(* Schneider Machine Expert - Basic project Tank_Level_RTD_1m_TM221CE40T, file version 3.0.0.0 *)
(* ProjectInformations: Name=New project *)

HARDWARE
  Cpu 0: TM221CE40T
  ModuleExtensionObject 0: TM3TI4/G
  EthernetConfiguration: NetworkName=M221, IpAllocationMode=FixedAddress, IpAddress=0.0.0.0, SubnetMask=0.0.0.0
  SerialLineConfiguration: Baud=Baud19200, Parity=ParityEven, DataBits=DataBits8, StopBits=StopBits1, PhysicalMedium=PhysicalMediumRs485, TransmissionMode=TransmissionModeModbusRtu, SlaveId=1, Addressing=SlaveAddressing
  MastTask: UsePeriodScanMode=false, PeriodScan=100
  FastTask: Period=255
  CpuBehavior: StartingMode=StartAsPreviousState, AutoSaveRamOnEeprom=true, WatchdogPeriod=250

SYMBOLS  (address, symbol, comment, settings)
  %M0       SYSTEM_READY
  %M1       TANK_FULL
  %M2       TANK_EMPTY
  %M3       FILLING_MODE
  %M4       DRAINING_MODE
  %M5       INLET_VLV_ALARM
  %M6       OUTLET_VLV_ALARM
  %M10      ANY_ALARM
  %S0       SB_COLDSTART  "Indicates or executes a cold start (data initialized to default values)"
  %S1       SB_WARMSTART  "Indicates there was a warm start with data backup"
  %MF102    HMI_TANK_LITERS  "HMI Tag: Tank volume in liters (0.0-1000.0) - scaled from %MW100"
  %MF103    HMI_TEMPERATURE  "HMI Tag: Temperature in degrees C - scaled from %MW101"
  %MF104    HMI_LEVEL_PERCENT  "HMI Tag: Level percentage (0.0-100.0) - calculated from %MF102"
  %TM1        [Preset=10, Base=OneSecond]
  %TM2        [Preset=5, Base=OneSecond]
  %TM3        [Preset=5, Base=OneSecond]
  %I0.0     EMERGENCY_PB
  %IW0.0      [Type=Type_0_10V, Scope=Scope_Normal, Minimum=0, Maximum=1000]
  %IW1.0    RTD_TEMP  [Type=Type_PT100, Scope=Scope_Standard, Minimum=-200, Maximum=850]

POU Tank Level Control
  (* SectionNumber=0 *)

// Rung 0: Reset_HMI
// Reset HMI floats on cold/warm start to prevent stale data display
  LD %S0                  (* SB_COLDSTART - Cold start *)
  OR %S1                  (* SB_WARMSTART - Warm start *)
  [ %MF102 := 0.0 ]       (* HMI_TANK_LITERS - Reset HMI Tank Liters *)
  [ %MF103 := 0.0 ]       (* HMI_TEMPERATURE - Reset HMI Temperature *)
  [ %MF104 := 0.0 ]       (* HMI_LEVEL_PERCENT - Reset HMI Level Percent *)
  // as ST:
  //   IF SB_COLDSTART OR SB_WARMSTART THEN HMI_TANK_LITERS := 0.0; END_IF;
  //   IF SB_COLDSTART OR SB_WARMSTART THEN HMI_TEMPERATURE := 0.0; END_IF;
  //   IF SB_COLDSTART OR SB_WARMSTART THEN HMI_LEVEL_PERCENT := 0.0; END_IF;
  (* the ladder stored for this rung does not match its IL; not drawn *)

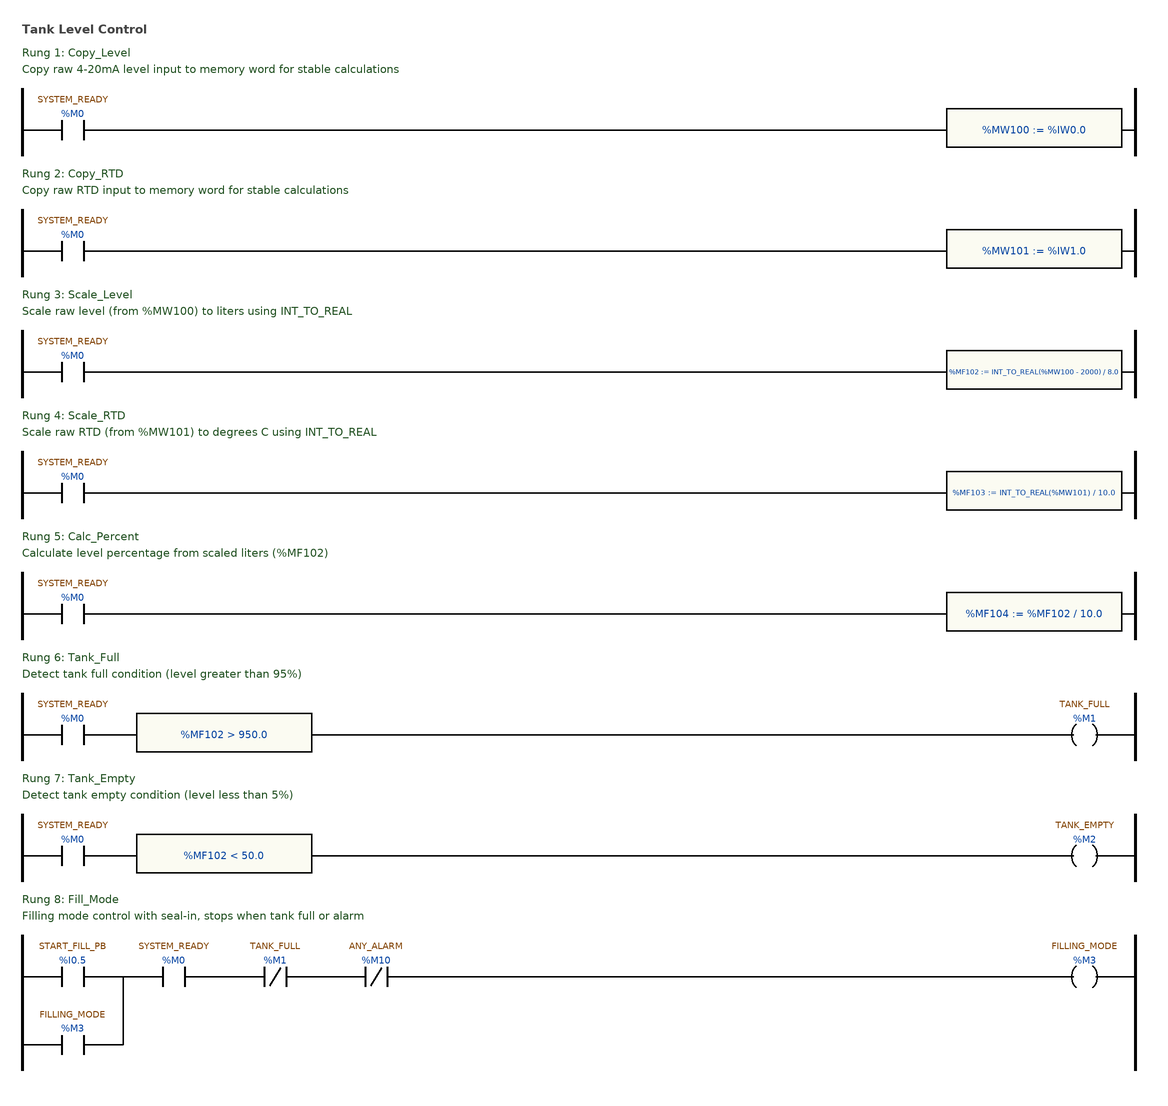

// Rung 1: Copy_Level
// Copy raw 4-20mA level input to memory word for stable calculations
  LD %M0                  (* SYSTEM_READY - System Ready *)
  [ %MW100 := %IW0.0 ]    (* Copy raw level to memory word *)
  // %M0: System Ready
  // as ST:
  //   IF SYSTEM_READY THEN %MW100 := %IW0.0; END_IF;

// Rung 2: Copy_RTD
// Copy raw RTD input to memory word for stable calculations
  LD %M0                  (* SYSTEM_READY - System Ready *)
  [ %MW101 := %IW1.0 ]    (* RTD_TEMP - Copy raw RTD to memory word *)
  // %M0: System Ready
  // as ST:
  //   IF SYSTEM_READY THEN %MW101 := RTD_TEMP; END_IF;

// Rung 3: Scale_Level
// Scale raw level (from %MW100) to liters using INT_TO_REAL
  LD %M0                  (* SYSTEM_READY - System Ready *)
  [ %MF102 := INT_TO_REAL(%MW100 - 2000) / 8.0 ](* HMI_TANK_LITERS - Scale 4-20mA to 0-1000.0 liters *)
  // %M0: System Ready
  // as ST:
  //   IF SYSTEM_READY THEN HMI_TANK_LITERS := INT_TO_REAL(%MW100 - 2000) / 8.0; END_IF;

// Rung 4: Scale_RTD
// Scale raw RTD (from %MW101) to degrees C using INT_TO_REAL
  LD %M0                  (* SYSTEM_READY - System Ready *)
  [ %MF103 := INT_TO_REAL(%MW101) / 10.0 ](* HMI_TEMPERATURE - Scale raw RTD to degrees C *)
  // %M0: System Ready
  // as ST:
  //   IF SYSTEM_READY THEN HMI_TEMPERATURE := INT_TO_REAL(%MW101) / 10.0; END_IF;

// Rung 5: Calc_Percent
// Calculate level percentage from scaled liters (%MF102)
  LD %M0                  (* SYSTEM_READY - System Ready *)
  [ %MF104 := %MF102 / 10.0 ](* HMI_LEVEL_PERCENT, HMI_TANK_LITERS - 0-1000 liters to 0-100.0 percent *)
  // %M0: System Ready
  // as ST:
  //   IF SYSTEM_READY THEN HMI_LEVEL_PERCENT := HMI_TANK_LITERS / 10.0; END_IF;

// Rung 6: Tank_Full
// Detect tank full condition (level greater than 95%)
  LD %M0                  (* SYSTEM_READY - System Ready *)
  AND [ %MF102 > 950.0 ]  (* HMI_TANK_LITERS - Level > 95% *)
  ST %M1                  (* TANK_FULL - Tank Full *)
  // %M0: System Ready
  // %M1: Tank Full Flag
  // as ST:
  //   TANK_FULL := SYSTEM_READY AND HMI_TANK_LITERS > 950.0;

// Rung 7: Tank_Empty
// Detect tank empty condition (level less than 5%)
  LD %M0                  (* SYSTEM_READY - System Ready *)
  AND [ %MF102 < 50.0 ]   (* HMI_TANK_LITERS - Level less than 5% *)
  ST %M2                  (* TANK_EMPTY - Tank Empty *)
  // %M0: System Ready
  // %M2: Tank Empty Flag
  // as ST:
  //   TANK_EMPTY := SYSTEM_READY AND HMI_TANK_LITERS < 50.0;

// Rung 8: Fill_Mode
// Filling mode control with seal-in, stops when tank full or alarm
  LD %I0.5                (* Start Fill Button *)
  OR %M3                  (* FILLING_MODE - Seal-in *)
  AND %M0                 (* SYSTEM_READY - System Ready *)
  ANDN %M1                (* TANK_FULL - Not Tank Full *)
  ANDN %M10               (* ANY_ALARM - No Alarm *)
  ST %M3                  (* FILLING_MODE - Filling Mode *)
  // %I0.5: Start Fill Button
  // %M0: System Ready
  // %M1: Not Tank Full
  // %M10: No Alarm
  // %M3: Filling Mode
  // %M3: Seal-in
  // as ST:
  //   FILLING_MODE := (%I0.5 OR FILLING_MODE) AND SYSTEM_READY AND NOT TANK_FULL AND NOT ANY_ALARM;

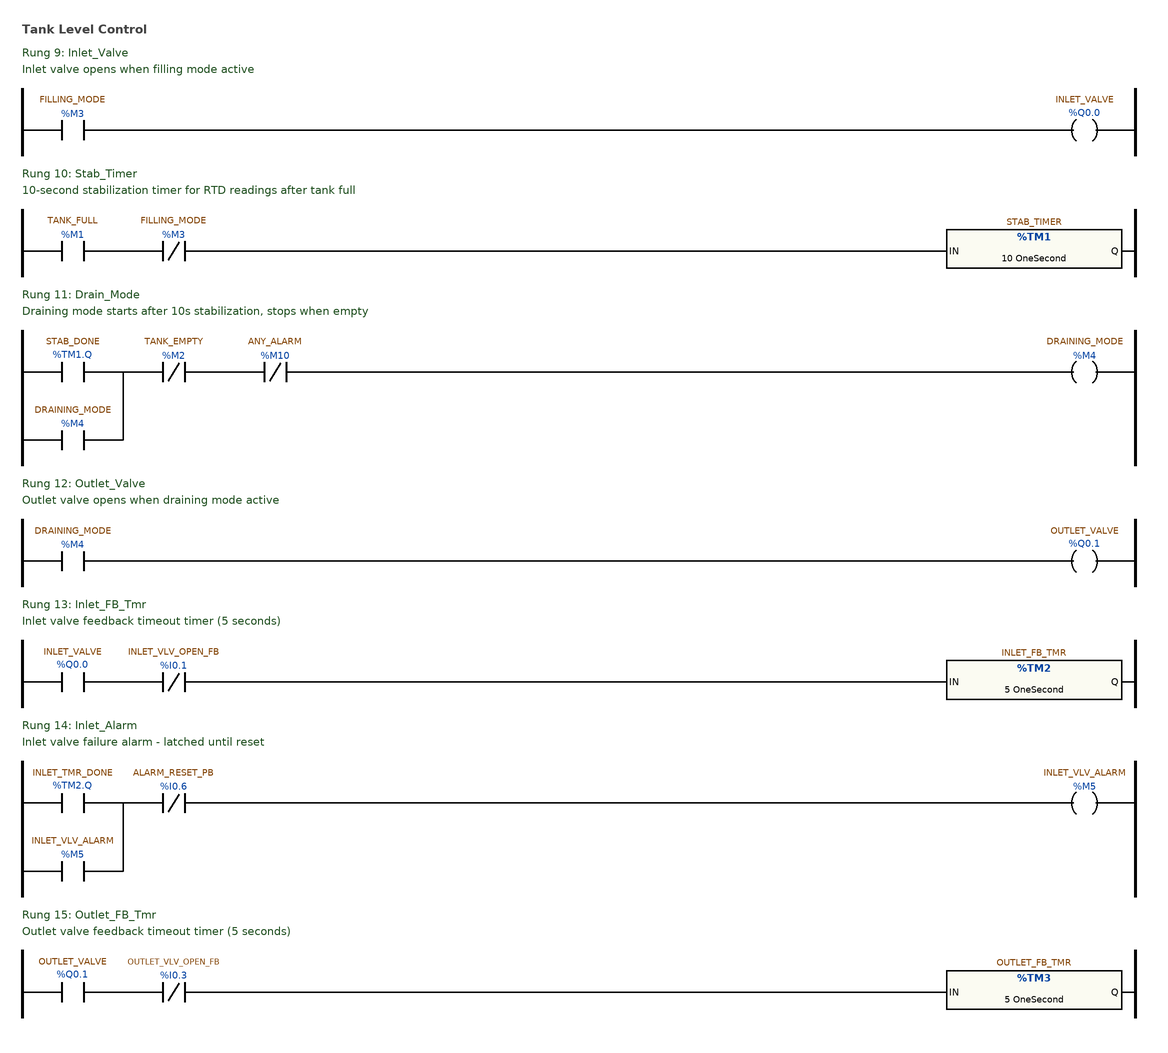

// Rung 9: Inlet_Valve
// Inlet valve opens when filling mode active
  LD %M3                  (* FILLING_MODE - Filling Mode *)
  ST %Q0.0                (* Open Inlet Valve *)
  // %M3: Filling Mode
  // %Q0.0: Inlet Valve
  // as ST:
  //   %Q0.0 := FILLING_MODE;

// Rung 10: Stab_Timer
// 10-second stabilization timer for RTD readings after tank full
  BLK %TM1                (* 10s Stabilization Timer *)
  LD %M1                  (* TANK_FULL - Tank Full *)
  ANDN %M3                (* FILLING_MODE - Filling Stopped *)
  IN
  OUT_BLK
  END_BLK
  // %M1: Tank Full
  // %M3: Filling Stopped
  // %TM1: 10s Stabilization
  // as ST:
  //   %TM1(IN := TANK_FULL AND NOT FILLING_MODE);

// Rung 11: Drain_Mode
// Draining mode starts after 10s stabilization, stops when empty
  LD %TM1.Q               (* 10s Timer Done *)
  OR %M4                  (* DRAINING_MODE - Seal-in *)
  ANDN %M2                (* TANK_EMPTY - Not Tank Empty *)
  ANDN %M10               (* ANY_ALARM - No Alarm *)
  ST %M4                  (* DRAINING_MODE - Draining Mode *)
  // %TM1.Q: Timer Done
  // %M2: Not Empty
  // %M10: No Alarm
  // %M4: Draining Mode
  // %M4: Seal-in
  // as ST:
  //   DRAINING_MODE := (%TM1.Q OR DRAINING_MODE) AND NOT TANK_EMPTY AND NOT ANY_ALARM;

// Rung 12: Outlet_Valve
// Outlet valve opens when draining mode active
  LD %M4                  (* DRAINING_MODE - Draining Mode *)
  ST %Q0.1                (* Open Outlet Valve *)
  // %M4: Draining Mode
  // %Q0.1: Outlet Valve
  // as ST:
  //   %Q0.1 := DRAINING_MODE;

// Rung 13: Inlet_FB_Tmr
// Inlet valve feedback timeout timer (5 seconds)
  BLK %TM2                (* Inlet Valve Feedback Timer *)
  LD %Q0.0                (* Inlet Valve Cmd *)
  ANDN %I0.1              (* No Open Feedback *)
  IN
  OUT_BLK
  END_BLK
  // %Q0.0: Inlet Cmd On
  // %I0.1: No Feedback
  // %TM2: 5s Feedback Timer
  // as ST:
  //   %TM2(IN := %Q0.0 AND NOT %I0.1);

// Rung 14: Inlet_Alarm
// Inlet valve failure alarm - latched until reset
  LD %TM2.Q               (* Timer Done *)
  OR %M5                  (* INLET_VLV_ALARM - Seal-in Alarm *)
  ANDN %I0.6              (* Reset Not Pressed *)
  ST %M5                  (* INLET_VLV_ALARM - Inlet Valve Alarm *)
  // %TM2.Q: Timer Done
  // %I0.6: Reset Not Pressed
  // %M5: Inlet Valve Alarm
  // %M5: Seal-in
  // as ST:
  //   INLET_VLV_ALARM := (%TM2.Q OR INLET_VLV_ALARM) AND NOT %I0.6;

// Rung 15: Outlet_FB_Tmr
// Outlet valve feedback timeout timer (5 seconds)
  BLK %TM3                (* Outlet Valve Feedback Timer *)
  LD %Q0.1                (* Outlet Valve Cmd *)
  ANDN %I0.3              (* No Open Feedback *)
  IN
  OUT_BLK
  END_BLK
  // %Q0.1: Outlet Cmd On
  // %I0.3: No Feedback
  // %TM3: 5s Feedback Timer
  // as ST:
  //   %TM3(IN := %Q0.1 AND NOT %I0.3);

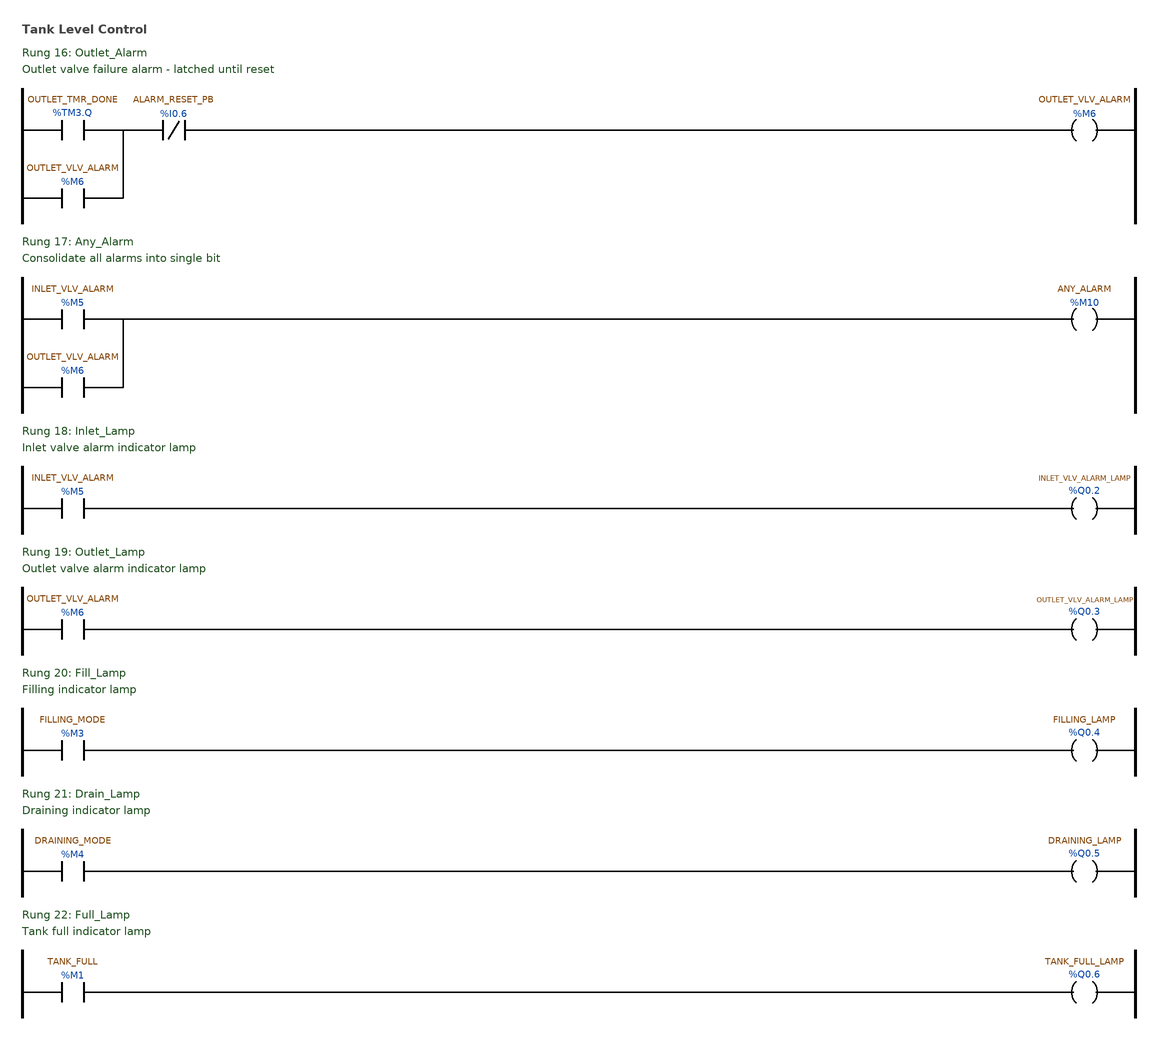

// Rung 16: Outlet_Alarm
// Outlet valve failure alarm - latched until reset
  LD %TM3.Q               (* Timer Done *)
  OR %M6                  (* OUTLET_VLV_ALARM - Seal-in Alarm *)
  ANDN %I0.6              (* Reset Not Pressed *)
  ST %M6                  (* OUTLET_VLV_ALARM - Outlet Valve Alarm *)
  // %TM3.Q: Timer Done
  // %I0.6: Reset Not Pressed
  // %M6: Outlet Valve Alarm
  // %M6: Seal-in
  // as ST:
  //   OUTLET_VLV_ALARM := (%TM3.Q OR OUTLET_VLV_ALARM) AND NOT %I0.6;

// Rung 17: Any_Alarm
// Consolidate all alarms into single bit
  LD %M5                  (* INLET_VLV_ALARM - Inlet Alarm *)
  OR %M6                  (* OUTLET_VLV_ALARM - Outlet Alarm *)
  ST %M10                 (* ANY_ALARM - Any Alarm *)
  // %M5: Inlet Alarm
  // %M10: Any Alarm
  // %M6: Outlet Alarm
  // as ST:
  //   ANY_ALARM := INLET_VLV_ALARM OR OUTLET_VLV_ALARM;

// Rung 18: Inlet_Lamp
// Inlet valve alarm indicator lamp
  LD %M5                  (* INLET_VLV_ALARM - Inlet Alarm *)
  ST %Q0.2                (* Inlet Alarm Lamp *)
  // %M5: Inlet Alarm
  // %Q0.2: Inlet Alarm Lamp
  // as ST:
  //   %Q0.2 := INLET_VLV_ALARM;

// Rung 19: Outlet_Lamp
// Outlet valve alarm indicator lamp
  LD %M6                  (* OUTLET_VLV_ALARM - Outlet Alarm *)
  ST %Q0.3                (* Outlet Alarm Lamp *)
  // %M6: Outlet Alarm
  // %Q0.3: Outlet Alarm Lamp
  // as ST:
  //   %Q0.3 := OUTLET_VLV_ALARM;

// Rung 20: Fill_Lamp
// Filling indicator lamp
  LD %M3                  (* FILLING_MODE - Filling Mode *)
  ST %Q0.4                (* Filling Lamp *)
  // %M3: Filling Mode
  // %Q0.4: Filling Lamp
  // as ST:
  //   %Q0.4 := FILLING_MODE;

// Rung 21: Drain_Lamp
// Draining indicator lamp
  LD %M4                  (* DRAINING_MODE - Draining Mode *)
  ST %Q0.5                (* Draining Lamp *)
  // %M4: Draining Mode
  // %Q0.5: Draining Lamp
  // as ST:
  //   %Q0.5 := DRAINING_MODE;

// Rung 22: Full_Lamp
// Tank full indicator lamp
  LD %M1                  (* TANK_FULL - Tank Full *)
  ST %Q0.6                (* Tank Full Lamp *)
  // %M1: Tank Full
  // %Q0.6: Tank Full Lamp
  // as ST:
  //   %Q0.6 := TANK_FULL;

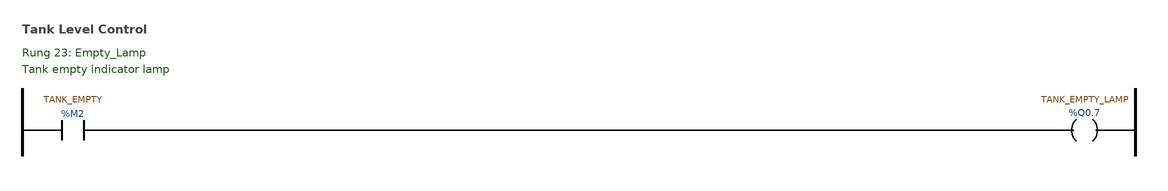

// Rung 23: Empty_Lamp
// Tank empty indicator lamp
  LD %M2                  (* TANK_EMPTY - Tank Empty *)
  ST %Q0.7                (* Tank Empty Lamp *)
  // %M2: Tank Empty
  // %Q0.7: Tank Empty Lamp
  // as ST:
  //   %Q0.7 := TANK_EMPTY;
